(* IEC 61131-3 sources: AXOpen/src/components.rexroth.drives/ctrl/src (part 4) *)

(* ---- AxoIndraDriveAxisData.st ---- *)
NAMESPACE AXOpen.Components.Rexroth.Drives
    CLASS AxoIndraDriveAxisData
        VAR PUBLIC
            (* Commands *)
            CallAxis					:	BOOL;			//Call axis method for cyclic communication
            ReadOnlyData				:	BOOL;			//Read only data values from drive
            CallNumberCyclic			:	INT :=-1; 		//Number of method call's for cyclic communication
            WriteCommand				:	BOOL;			//Write command to drive
            PowerOnReq					:	BOOL;			//Request to power the drive on
            ResetReq					:	BOOL;			//Request to reset the drive
            HomingReq					:	BOOL;			//Request to start homing
            JogPositiveReq				:	BOOL;			//Request to jog the drive in positive direction
            JogNegativeReq				:	BOOL;			//Request to jog the drive in negative direction
            DriveStopReq				:	BOOL;			//Set Drive Stop with writing deceleration value to drive
            DriveHaltReq				:	BOOL;			//Set Drive Halt with writing deceleration value to drive
            MoveVelocityReq				:	BOOL;			//Command is velocity
            TorqueControlReq				:	BOOL;			//Command is torque
            Relative					:	BOOL; 			//Move relative to (last recommended) positioning command value
            Additive					:	BOOL; 			//Move additive to actual position; works only if relative possitioning active
            Position					:	LREAL;			//Target position for the motion  (negative or positive)
            Velocity					:	LREAL;			//Value of the maximum velocity (always positive) (not necessarily reached) [u/s].
            Acceleration				:	LREAL;			//Value of the acceleration (always positive) (increasing energy of the motor) [u/s2]
            Deceleration				:	LREAL;			//Value of the deceleration (always positive) (decreasing energy of the motor) [u/s2]
            Jerk						:	LREAL;			//Value of the jerk (always positive) [u/s3]
            Torque						:	LREAL;			//Value of the torque (always positive)
            S_0_0144_SignalStateWord	: 	WORD;			//S-0-0144 SignalStateWord*)
            CallAxisParameterMethod		:	BOOL;			//Call axis method for parameter read/write
            EnableAcyclicCommunication	:	BOOL;			//Enable acyclic communication (for parameter read/write)
            CallNumberAcyclic			:	INT;			//Number of method call's for acyclic communication
            WriteParameter				:	BOOL;			//FALSE = read, TRUE  = write Value of selected Parameter
            SelectDataType				:	UINT;			//0= Bool, 1 = Any, 2 = REAL
            ParameterNumber				:	DINT;			//Parameter number
            WriteValueDint				:	DINT;			//DINT value to be written
            WriteValueReal				:	REAL;			//REAL value to be written
            OverrideVelocityFactor		:	LREAL := 1.0;	//LREAL value to be written
            OverrideAccelerationFactor	:	LREAL := 1.0;	//LREAL value to be written
            OverrideJerkFactor			:	LREAL := 1.0;	//LREAL value to be written
        (* States *)
            CommandWriteActive			:	BOOL; 			//Command transfer to drive is active
            SetpointReached				: 	BOOL;			//Setpoint reached
            PowerOK						:	BOOL; 			//Power OK
            HomeOK						:	BOOL;			//Drive has reached the homeposition
            ResetOK						:	BOOL; 			//Reset done
            HomingRunning				:	BOOL;			//Homing is active
            Stopped						:	BOOL; 			//Drive in stopped regularly
            Standstill					:	BOOL; 			//Drive in standstill
            InPosition					:	BOOL; 			//Drive in position
            StoppedDueError				:	BOOL; 			//Drive in stop due to error
            MessageActive				:	BOOL;			//Class 3 diagnostics (message) present
            WarningActive				:	BOOL;			//Class 2 diagnostics (warning) present
            FailureActive				:	BOOL;			//Class 1 diagnostics (failure) present
            PowerError					:	BOOL; 			//Power-Failure
            StopError					:	BOOL;			//Stopping-Failure
            ContinuousMotion			:	BOOL; 			//Continius motion
            DiscreteMotion				:	BOOL; 			//Discrete motion
            SynchronizedMotion			:	BOOL;			//Synchronized motion
            Error						:	BOOL;			//Error
            ErrorID						:	AXOpen.Components.Rexroth.Drives.eAxoIndraDriveErrorCode;		//Error identification, ErrorCode
            ErrorIdent					:	AXOpen.Components.Rexroth.Drives.AxoIndraDriveErrorStruct;	//Error identification
            ActualPosition				:	LREAL; 			//Shows actual position
            ActualVelocity				:	LREAL; 			//Shows actual velocity
            ActualTorque				:	LREAL; 			//Shows actual torque
            CheckAccessOK				:	BOOL := TRUE;	//Flag for checking valid access at Axis_Data array
            S_0_0145_SignalControlWord	:	WORD;			//S-0-0145 wSignalControlWord, **** exept bit 0 *****)

            DoneAcyclicCommunication 	:	BOOL; 			//Reading/writing of the individual parameter completed, output variables valid
            ActiveAcyclicCommunication	: 	BOOL; 			//Reading/writing of the individual parameter active, output variables invalid
            DecimalPlaces 				:	UINT;			//Decimal places of the selected parameters
            DataTypeRead				:	UINT; 			//Read data type of the selected parameters
            DataLengthRead				:	UINT;			//Length of the read parameters
            ReadValueDint				:	DINT;			//DINT Operating value of the individual parameter without weighting
            ReadValueReal				:	REAL;			//REAL weighted operating value
            Error_AcyclicCommunication	:	BOOL := FALSE;  //Error
            ErrorID_AcyclicCommunication:   AXOpen.Components.Rexroth.Drives.eAxoIndraDriveErrorCode;		//Error identification, ErrorCode
            ErrorIdent_AcyclicCommunication:AXOpen.Components.Rexroth.Drives.AxoIndraDriveErrorStruct; 	//Error identification

        END_VAR

    END_CLASS

END_NAMESPACE

(* ---- AxoIndraDriveAxisReference.st ---- *)
// USING AXOpen.Components.Drives;

NAMESPACE AXOpen.Components.Rexroth.Drives
    CLASS AxoIndraDriveAxisReference IMPLEMENTS AXOpen.Components.Abstractions.Drives.IAxoAxisReference
        VAR PUBLIC
            FieldBus_In     :   AXOpen.Components.Rexroth.Drives.AxoIndraDriveFieldBusIn;
            FieldBus_Out    :   AXOpen.Components.Rexroth.Drives.AxoIndraDriveFieldBusOut;
            Parameter_In    :   AXOpen.Components.Rexroth.Drives.AxoIndraDriveParameterIn;
            Parameter_Out   :   AXOpen.Components.Rexroth.Drives.AxoIndraDriveParameterOut;
            Data            :   AXOpen.Components.Rexroth.Drives.AxoIndraDriveAxisData;
            Config          :   AXOpen.Components.Drives.AxoDrive_Config;
            Status          :   AXOpen.Components.Drives.AxoDrive_Status;
        END_VAR
    END_CLASS
END_NAMESPACE

(* ---- AxoIndraDriveFieldBusIn.st ---- *)
NAMESPACE AXOpen.Components.Rexroth.Drives
    CLASS AxoIndraDriveFieldBusIn
        (******************* Drive configuration  ***********************
        Master communication; Fieldbus settings:

                Profile type: * free configurable mode*
                    Configuration of realtime channel:
                        realtime input (configured feedback values):	    (9words)
                                P-0-4078 Fieldbus status WORD               (2bytes)
                                S-0-0051 Position feedback 1 value          (4bytes)
                                S-0-0040 Veloccity feedback value           (4bytes)
                                S-0-0390 Diagnostig message number          (4bytes)
                                S-0-0144 Signal status  word			    (2bytes)
                                S-0-0084 Actual torque/force value          (2bytes)
                        realtime output (configured command values):		(13words)
                                P-0-4077 Fieldbus control WORD              (2bytes)
                                S-0-0282 Positioning command value          (4bytes)
                                S-0-0259 Positioning velocity value         (4bytes)
                                S-0-0260 Positioning Accelelration          (4bytes)
                                S-0-0359 Positioning Deceleration           (4bytes)
                                S-0-0145 Signal control word                (2bytes)
                                S-0-0080 Torque/force command value		    (2bytes)
                                S-0-0193 Positioning jerk                   (4bytes)
                General settings:
                        S-0-0027, Configuration list signal control word -> Number 0; Content S-0-0393
                        S-0-0329, Assign list signal control word -> Number 0; Content 2
                        Primary operation mode: Drive controlled positioning, encoder 1 (without axis control word)
                        Secondary operation mode: Torque/force control
        *)
        VAR PUBLIC
            PhaseAcknowledgeBit0		:	BOOL;		//Operating mode acknowledge bit 0
            PhaseAcknowledgeBit1 		:	BOOL;		//Operating mode acknowledge bit 1
            InReference 				:	BOOL;		//In reference
            InStandstill 				:	BOOL;		//In standstill
            SetpointReached				:	BOOL;		//Setpoint reached
            CommandChangeBit 			:	BOOL;		//Command change bit
            OperatingModeError 			:	BOOL;		//Operating mode_error
            StatusSetpointProcess 		:	BOOL;		//Status setpoint processing
            ActualOperatingModeBit0 	:	BOOL;		//Actual_operating mode bit 0
            ActualOperatingModeBit1 	:	BOOL;		//Actual_operating mode bit 1
            SetpointAcknowledge 		:	BOOL;		//Setpoint acknowledge
            MessageZKL3 				:	BOOL;		//Message ZKL3
            WarningZKL2 				:	BOOL;		//Warning ZKL2
            DriveErrorZKL1 				:	BOOL;		//Drive Error ZKL1
            ReadyToOperateBit0 			:	BOOL;		//Ready to operate bit 0
            ReadyToOperateBit1 			:	BOOL;		//Ready to operate bit 1
            S_0_0051_ActualPosition		:	DWORD;		//Actual position
            S_0_0040_ActualVelocity		:	DWORD;		//Actual velocity
            S_0_0390_Diagnosis			:	DWORD;		//Diagnosis
            S_0_0144_SignalStatusWord	:	WORD;		//Signal status word
            S_0_0084_ActualTorque 		:	WORD;		//Actual torque
        END_VAR
    END_CLASS

END_NAMESPACE

(* ---- AxoIndraDriveFieldBusOut.st ---- *)
NAMESPACE AXOpen.Components.Rexroth.Drives
    CLASS AxoIndraDriveFieldBusOut
        (******************* Drive configuration  ***********************
        Master communication; Fieldbus settings:

                Profile type: * free configurable mode*
                    Configuration of realtime channel:
                        realtime input (configured feedback values):	    (9words)
                                P-0-4078 Fieldbus status WORD               (2bytes)
                                S-0-0051 Position feedback 1 value          (4bytes)
                                S-0-0040 Veloccity feedback value           (4bytes)
                                S-0-0390 Diagnostig message number          (4bytes)
                                S-0-0144 Signal status  word			    (2bytes)
                                S-0-0084 Actual torque/force value          (2bytes)
                        realtime output (configured command values):		(13words)
                                P-0-4077 Fieldbus control WORD              (2bytes)
                                S-0-0282 Positioning command value          (4bytes)
                                S-0-0259 Positioning velocity value         (4bytes)
                                S-0-0260 Positioning Accelelration          (4bytes)
                                S-0-0359 Positioning Deceleration           (4bytes)
                                S-0-0145 Signal control word                (2bytes)
                                S-0-0080 Torque/force command value		    (2bytes)
                                S-0-0193 Positioning jerk                   (4bytes)
                General settings:
                        S-0-0027, Configuration list signal control word -> Number 0; Content S-0-0393
                        S-0-0329, Assign list signal control word -> Number 0; Content 2
                        Primary operation mode: Drive controlled positioning, encoder 1 (without axis control word)
                        Secondary operation mode: Torque/force control
        *)
        VAR PUBLIC
            SetpointAcceptance 				:	BOOL;			//Setpoint acceptance
            OperatingModeSet 				:	BOOL;			//Operating mode set
            DriveToZeroPoint 				:	BOOL;			//Drive to zero point
            AbsoluteRelative 				:	BOOL;			//Position absolute = 0 or relative = 1
            ImmediateBlockChange 			:	BOOL;			//Immediate change
            ErrorDelete 					:	BOOL;			//Clear error
            JogForward 						:	BOOL;			//Jog forward
            JogBackward 					:	BOOL;			//Jog backward
            SetOperatingModeBit0 			:	BOOL;			//Setpoint operating mode_bit0
            SetOperatingModeBit1 			:	BOOL;			//Setpoint operating mode_bit1
            Iposync 						:	BOOL;			//Only in cycl. pos. control
            DriveHalt 						:	BOOL;			//Drive halt
            DriveEnable 					:	BOOL;			//Drive enable
            DriveOn 						:	BOOL;			//Drive on
            S_0_0282_CommandPosition		: 	DWORD;			//Command position
            S_0_0259_CommandVelocity		: 	DWORD;          //Command velocity
            S_0_0260_CommandAcceleration	: 	DWORD;          //Command acceleration
            S_0_0359_CommandDecceleration	: 	DWORD;          //Command decceleration
            S_0_0145_SignalControlWord		: 	WORD;           //Signal control word
            S_0_0080_TorqueForceCommand     :   WORD;           //Torque/force command value
            S_0_0193_CommandJerk            :   DWORD;          //Command jerk
        END_VAR
    END_CLASS
END_NAMESPACE

(* ---- AxoIndraDriveParameterIn.st ---- *)
NAMESPACE AXOpen.Components.Rexroth.Drives
    CLASS AxoIndraDriveParameterIn
        (******************* IndraDrive configuration  ***********************
        Master communication; Fieldbus settings:
        Parameter chanel 10Bytes / 5 Words I/O
        *)
        VAR PUBLIC
            Datalength	:	BYTE;	//Length of  transfer data*)
            FL_0		:	BOOL;	//Length userdata bit 0
            FL_1		:	BOOL;	//Length userdata bit 1
            FL_2		:	BOOL;	//Length userdata bit 2
            FL_3		:	BOOL;	//Length userdata bit 3
            ToggleBit	:	BOOL;	//Toggle bit
            LastBit		:	BOOL;	//Last bit
            Failure		:	BOOL;	//Failure while communication
            Reserve		:	BOOL;	//Reserve
            DataWord_0	:	WORD;	//Data WORD 0
            DataWord_1	:	WORD;	//Data word 1
            DataWord_2	:	WORD;	//Data word 2
            DataWord_3	:	WORD;	//Data word 3
        END_VAR
    END_CLASS
 END_NAMESPACE

(* ---- AxoIndraDriveParameterOut.st ---- *)
NAMESPACE AXOpen.Components.Rexroth.Drives
    CLASS AxoIndraDriveParameterOut
        (******************* IndraDrive configuration  ***********************
        Master communication; Fieldbus settings:
        Parameter chanel 10Bytes / 5 Words I/O
        *)
        VAR PUBLIC
            Datalength		:	BYTE := BYTE#04;//Length of transfer data
            FL_0			:	BOOL;			//Length userdata bit 0
            FL_1			:	BOOL;			//Length userdata bit 1
            FL_2			:	BOOL;			//Length userdata bit 2
            FL_3			:	BOOL;			//Length userdata bit 3
            ToggleBit		:	BOOL;			//Toggle bit
            LastBit			:	BOOL;			//Last bit
            Initalisation	:	BOOL := TRUE;	//Initialisation
            Reserve			:	BOOL;			//Reserve
            Index			:	WORD;			//Index number
            Subindex		:	BYTE;			//Subindex number
            Axis			:	BYTE;			//Axis number
            DataWord_0		:	WORD;			//Data word 0
            DataWord_1		:	WORD;			//Data word 1
        END_VAR
    END_CLASS
END_NAMESPACE

(* ---- AxoRexrothDrive.st ---- *)
USING AXOpen.Messaging.Static;
USING AXOpen.Messaging;
USING AXOpen.Core;
USING AXOpen.Components.Abstractions;
USING AXOpen.Components.Abstractions.AxoDrives;

NAMESPACE AXOpen.Components.Rexroth.Drives
    {#ix-attr:[Container(Layout.Wrap)]}
    CLASS PUBLIC AxoIndraDrive EXTENDS AXOpen.Components.Abstractions.AxoDrives.AxoDrive IMPLEMENTS AXOpen.Components.Abstractions.AxoDrives.IAxoDrive
        VAR PUBLIC
        END_VAR

        ///<summary>
		/// Restores this instance .
        ///</summary>
        METHOD PROTECTED OVERRIDE Restore: IAxoTask
            VAR
                _index : INT;
            END_VAR
            // Status.Action.Id := UINT#0;
            // Status.Error.Id  := UINT#0;
            // Status.CurrentJobName := '';
            // _Messenger.Restore();
            // _TaskMessenger.Restore();

            // ClearInspectionResultsTask.Restore();
            // TriggerTask.Restore();
            // ChangeJobByNameTask.Restore();
            // ChangeJobByNumberTask.Restore();

            // IF NOT AcquisitionStatus.ExposureComplete AND NOT InspectionStatus.Error THEN
            //     Status.Action.Id := UINT#300;
            //     RestoreTask.DoneWhen(TRUE);
            // END_IF;
            ;
        END_METHOD

        ///<summary>
		/// Custom logic for the manual control.
        ///</summary>
        METHOD PROTECTED OVERRIDE ManualControl
            // ChangeJobByNameTask.Manual(RequiredJobName);
            // ChangeJobByNumberTask.Manual(RequiredJobNumber);
            // SoftEventTask.Manual(RequiredSoftEventNumber);
            ;
        END_METHOD

        ///<summary>
        /// Ensures swapping the hardware input data structure into the AxisRef data structure
        ///</summary>
        METHOD PROTECTED OVERRIDE UpdateInputs : BOOL
            VAR_INPUT
                refAxisIn       :   REF_TO  ARRAY[*] OF BYTE;   //  Reference to the input data of the axis
            END_VAR
            VAR_IN_OUT
                AxisRef    :   AxoAxisRef;
            END_VAR
            ;
        END_METHOD

        ///<summary>
        /// Ensures swapping the AxisRef data structure into the hardware output data structure
        ///</summary>
        METHOD PROTECTED OVERRIDE UpdateOutputs : BOOL
            VAR_IN_OUT
                AxisRef    :   AxoAxisRef;
            END_VAR
            VAR_INPUT
                refAxisOut      :   REF_TO  ARRAY[*] OF BYTE;   //  Reference to the output data of the axis
            END_VAR
            ;
        END_METHOD

        ///<summary>
        /// This method controls the power stage (On or Off).
        ///</summary>
        METHOD PUBLIC OVERRIDE MC_Power
            VAR_IN_OUT
                AxisRef         :   AxoAxisRef;
            END_VAR
            VAR_INPUT
                Enable          :   BOOL;                       //  As long as ‘Enable’ is true, power is being enabled.
            END_VAR
            VAR_OUTPUT
                Status          :   BOOL;                       //  Effective state of the power stage
                Valid           :   BOOL;                       //  If true, a valid set of outputs is available at the method
                Error           :   BOOL;                       //  Signals that an error has occurred within the method
                ErrorID         :   WORD;                       //  Error identification
            END_VAR
            ;
        END_METHOD

        ///<summary>
        /// This method commands the axis to perform the «search home» sequence. The details of this sequence are
        /// manufacturer dependent and can be set by the axis’ parameters. The ‘Position’ input is used to set the absolute
        /// position when reference signal is detected. This method completes at ‘Standstill’ if it was started in ‘Standstill’.
        ///</summary>
        METHOD PUBLIC OVERRIDE MC_Home
            VAR_IN_OUT
                AxisRef         :   AxoAxisRef;                 //  Reference to the axis
            END_VAR
            VAR_INPUT
                Execute         :   BOOL;                       //  Start the motion at rising edge
                Position        :   LREAL;                      //  Absolute position when the reference signal is detected
                HommingMode     :   INT;                        //  Required homming mode
                Velocity        :   LREAL;                      //  Value of the maximum ‘Velocity’ (not necessarily reached) [u/s].
                Acceleration    :   LREAL;                      //  Value of the ‘Acceleration’ (always positive) (increasing energy of the motor) [u/s2]
                Deceleration    :   LREAL;                      //  Value of the ‘Deceleration’ (always positive) (decreasing energy of the motor) [u/s2]
            END_VAR
            VAR_OUTPUT
                Done            :   BOOL;                       // Reference known and set sucessfully
                Busy            :   BOOL;                       // The method is not finished and new output values are to be expected
                Active          :   BOOL;                       // Indicates that the method has control on the axis
                CommandAborted  :   BOOL;                       // ‘Command’ is aborted by another command
                Error           :   BOOL;                       // Signals that an error has occurred within the method
                ErrorID         :   WORD;                       // Error identification
             END_VAR
             ;
        END_METHOD

        ///<summary>
        /// This method commands a controlled motion stop and transfers the axis to the state ‘Stopping’. It aborts any
        /// ongoing method execution. While the axis is in state ‘Stopping’, no other method can perform any motion on the
        /// same axis.
        ///</summary>
        METHOD PUBLIC OVERRIDE MC_Stop
            VAR_IN_OUT
                AxisRef         :   AxoAxisRef;                 //  Reference to the axis
            END_VAR
            VAR_INPUT
                Execute         :   BOOL;                       //  Start the action at rising edge
                Deceleration    :   LREAL;                      //  Value of the ‘Deceleration’ [u/s2]
                Jerk            :   LREAL;                      //  Value of the ‘Jerk’ [u/s3]
            END_VAR
            VAR_OUTPUT
                Done            :   BOOL;                       // Zero velocity reached
                Busy            :   BOOL;                       // The method is not finished and new output values are to be expected
                Active          :   BOOL;                       // Indicates that the method has control on the axis
                CommandAborted  :   BOOL;                       // ‘Command’ is aborted by switching off power (only possibility to abort)
                Error           :   BOOL;                       // Signals that an error has occurred within the method
                ErrorID         :   WORD;                       // Error identification
             END_VAR
             ;
        END_METHOD

        ///<summary>
        /// This method commands a controlled motion stop. The axis is moved to the state ‘DiscreteMotion’, until the
        /// velocity is zero. With the ‘Done’ output set, the state is transferred to ‘Standstill’.
        ///</summary>
        METHOD PUBLIC OVERRIDE MC_Halt
            VAR_IN_OUT
                AxisRef         :   AxoAxisRef;                 //  Reference to the axis
            END_VAR
            VAR_INPUT
                Execute         :   BOOL;                       //  Start the action at rising edge
                Deceleration    :   LREAL;                      //  Value of the ‘Deceleration’ [u/s2]
                Jerk            :   LREAL;                      //  Value of the ‘Jerk’ [u/s3]
            END_VAR
            VAR_OUTPUT
                Done            :   BOOL;                       // Zero velocity reached
                Busy            :   BOOL;                       // The method is not finished and new output values are to be expected
                Active          :   BOOL;                       // Indicates that the method has control on the axis
                CommandAborted  :   BOOL;                       // ‘Command’ is aborted by switching off power (only possibility to abort)
                Error           :   BOOL;                       // Signals that an error has occurred within the method
                ErrorID         :   WORD;                       // Error identification
             END_VAR
             ;
        END_METHOD

        ///<summary>
        /// This method commands a controlled motion to a specified absolute position.
        ///<summary>
        METHOD PUBLIC OVERRIDE MC_MoveAbsolute
            VAR_IN_OUT
                AxisRef         :   AxoAxisRef;                 //  Reference to the axis
            END_VAR
            VAR_INPUT
                Execute         :   BOOL;                       //  Start the motion at rising edge
                ContinuousUpdate:   BOOL;                       //  Activate ‘ContinuousUpdate’ - target parameters should be changed during movement
                Position        :   LREAL;                      //  Commanded ‘Position’ for the motion (in technical unit [u]) (negative or positive)
                Velocity        :   LREAL;                      //  Value of the maximum ‘Velocity’ (not necessarily reached) [u/s].
                Acceleration    :   LREAL;                      //  Value of the ‘Acceleration’ (always positive) (increasing energy of the motor) [u/s2]
                Deceleration    :   LREAL;                      //  Value of the ‘Deceleration’ (always positive) (decreasing energy of the motor) [u/s2]
                Jerk            :   LREAL;                      //  Value of the ‘Jerk’ [u/s3]
                Direction       :   eAxoDriveDirection;         //  Enum type (1-of-4 values: PositiveDirection, ShortestWay, NegativeDirection, CurrentDirection)
            END_VAR
            VAR_OUTPUT
                Done            :   BOOL;                       // Commanded position finally reached
                Busy            :   BOOL;                       // The method is not finished and new output values are to be expected
                Active          :   BOOL;                       // Indicates that the method has control on the axis
                CommandAborted  :   BOOL;                       // ‘Command’ is aborted by another command
                Error           :   BOOL;                       // Signals that an error has occurred within the method
                ErrorID         :   WORD;                       // Error identification
             END_VAR
             ;
        END_METHOD

        ///<summary>
        /// This method  commands a controlled motion of a specified distance relative to the set position at the time of the execution.
        ///<summary>
        METHOD PUBLIC OVERRIDE MC_MoveRelative
            VAR_IN_OUT
                AxisRef         :   AxoAxisRef;                 //  Reference to the axis
            END_VAR
            VAR_INPUT
                Execute         :   BOOL;                       //  Start the motion at rising edge
                ContinuousUpdate:   BOOL;                       //  Activate ‘ContinuousUpdate’ - target parameters should be changed during movement
                Distance        :   LREAL;                      //  Relative distance for the motion (in technical unit [u]
                Velocity        :   LREAL;                      //  Value of the maximum ‘Velocity’ (not necessarily reached) [u/s].
                Acceleration    :   LREAL;                      //  Value of the ‘Acceleration’ (always positive) (increasing energy of the motor) [u/s2]
                Deceleration    :   LREAL;                      //  Value of the ‘Deceleration’ (always positive) (decreasing energy of the motor) [u/s2]
                Jerk            :   LREAL;                      //  Value of the ‘Jerk’ [u/s3]
                Direction       :   eAxoDriveDirection;         //  Enum type (1-of-4 values: PositiveDirection, ShortestWay, NegativeDirection, CurrentDirection)
            END_VAR
            VAR_OUTPUT
                Done            :   BOOL;                       // Commanded distance reached
                Busy            :   BOOL;                       // The method is not finished and new output values are to be expected
                Active          :   BOOL;                       // Indicates that the method has control on the axis
                CommandAborted  :   BOOL;                       // ‘Command’ is aborted by another command
                Error           :   BOOL;                       // Signals that an error has occurred within the method
                ErrorID         :   WORD;                       // Error identification
             END_VAR
             ;
        END_METHOD

        ///<summary>
        /// This method commands a controlled motion of a specified relative distance additional to the most recent
        /// commanded position in the axis state ‘DiscreteMotion’. The most recent commanded position may be the result of a
        /// previous MC_MoveAdditive motion which was aborted. If the method is activated in the axis state ‘ContinuousMotion’, the
        /// specified relative distance is added to the set position at the time of the execution.
        ///<summary>
        METHOD PUBLIC OVERRIDE MC_MoveAdditive
            VAR_IN_OUT
                AxisRef         :   AxoAxisRef;                 //  Reference to the axis
            END_VAR
            VAR_INPUT
                Execute         :   BOOL;                       //  Start the motion at rising edge
                ContinuousUpdate:   BOOL;                       //  Activate ‘ContinuousUpdate’ - target parameters should be changed during movement
                Distance        :   LREAL;                      //  Relative distance for the motion (in technical unit [u]
                Velocity        :   LREAL;                      //  Value of the maximum ‘Velocity’ (not necessarily reached) [u/s].
                Acceleration    :   LREAL;                      //  Value of the ‘Acceleration’ (always positive) (increasing energy of the motor) [u/s2]
                Deceleration    :   LREAL;                      //  Value of the ‘Deceleration’ (always positive) (decreasing energy of the motor) [u/s2]
                Jerk            :   LREAL;                      //  Value of the ‘Jerk’ [u/s3]
                Direction       :   eAxoDriveDirection;         //  Enum type (1-of-4 values: PositiveDirection, ShortestWay, NegativeDirection, CurrentDirection)
            END_VAR
            VAR_OUTPUT
                Done            :   BOOL;                       // Commanded distance reached
                Busy            :   BOOL;                       // The method is not finished and new output values are to be expected
                Active          :   BOOL;                       // Indicates that the method has control on the axis
                CommandAborted  :   BOOL;                       // ‘Command’ is aborted by another command
                Error           :   BOOL;                       // Signals that an error has occurred within the method
                ErrorID         :   WORD;                       // Error identification
             END_VAR
             ;
        END_METHOD

        ///<summary>
        /// This method commands a never ending controlled motion at a specified velocity.
        ///<summary>
        METHOD PUBLIC OVERRIDE MC_MoveVelocity
            VAR_IN_OUT
                AxisRef         :   AxoAxisRef;                 //  Reference to the axis
            END_VAR
            VAR_INPUT
                Execute         :   BOOL;                       //  Start the motion at rising edge
                ContinuousUpdate:   BOOL;                       //  Activate ‘ContinuousUpdate’ - target parameters should be changed during movement
                Velocity        :   LREAL;                      //  Value of the maximum velocity [u/s]. Can be a signed value.
                Acceleration    :   LREAL;                      //  Value of the ‘Acceleration’ (always positive) (increasing energy of the motor) [u/s2]
                Deceleration    :   LREAL;                      //  Value of the ‘Deceleration’ (always positive) (decreasing energy of the motor) [u/s2]
                Jerk            :   LREAL;                      //  Value of the ‘Jerk’ [u/s3]
                Direction       :   eAxoDriveDirection;         //  Enum type (1-of-3 values: PositiveDirection, NegativeDirection, and CurrentDirection. Note: shortest way not applicable)
            END_VAR
            VAR_OUTPUT
                InVelocity      :   BOOL;                       // Commanded velocity reached
                Busy            :   BOOL;                       // The method is not finished and new output values are to be expected
                Active          :   BOOL;                       // Indicates that the method has control on the axis
                CommandAborted  :   BOOL;                       // ‘Command’ is aborted by another command
                Error           :   BOOL;                       // Signals that an error has occurred within the method
                ErrorID         :   WORD;                       // Error identification
             END_VAR
             ;
        END_METHOD

        ///<summary>
        /// This method continuously exerts a torque or force of the specified magnitude. This magnitude is
        /// approached using a defined ramp (‘TorqueRamp’), and the method sets the ‘InTorque’ output if the
        /// commanded torque level is reached. This method is applicable for force and torque. When there is no external
        /// load, force is applicable. Positive torque is in the positive direction of velocity.
        ///<summary>
        METHOD PUBLIC OVERRIDE MC_TorqueControl
            VAR_IN_OUT
                AxisRef         :   AxoAxisRef;                 //  Reference to the axis
            END_VAR
            VAR_INPUT
                Execute         :   BOOL;                       //  Start the motion at rising edge
                ContinuousUpdate:   BOOL;                       //  Activate ‘ContinuousUpdate’ - target parameters should be changed during movement
                Torque          :   LREAL;                      //  Value of the torque (Torque or force in technical unit [u])
                TorqueRamp      :   LREAL;                      //  The maximum time derivative of the set value of the torque or force (in technical unit per sec. [u/s])
                Velocity        :   LREAL;                      //  Absolute value of the maximum velocity.
                Acceleration    :   LREAL;                      //  Value of the maximum acceleration (acceleration is applicable with same sign of torque and velocity)
                Deceleration    :   LREAL;                      //  Value of the maximum deceleration (deceleration is applicable with opposite signs of torque and velocity)
                Jerk            :   LREAL;                      //  Value of the maximum jerk
                Direction       :   eAxoDriveDirection;         //  Enum type (1 of 2 values: PositiveDirection, NegativeDirection or CurrentDirection). Specifies the direction of the torque. (Note: Torque input can be signed value).
            END_VAR
            VAR_OUTPUT
                InTorque        :   BOOL;                       //  Setpoint value of torque or force equals the commandedvalue
                Busy            :   BOOL;                       //  The method is not finished and new output values are to be expected
                Active          :   BOOL;                       //  Indicates that the method has control on the axis
                CommandAborted  :   BOOL;                       //  ‘Command’ is aborted by another command
                Error           :   BOOL;                       //  Signals that an error has occurred within the method
                ErrorID         :   WORD;                       //  Error identification
            END_VAR
            ;
        END_METHOD

        ///<summary>
        /// This method shifts the coordinate system of an axis by manipulating both the set-point position as well as the
        /// actual position of an axis with the same value without any movement caused. (Re-calibration with same following error).
        /// This can be used for instance for a reference situation. This method can also be used during motion without changing
        /// the commanded position, which is now positioned in the shifted coordinate system.
        ///<summary>
        METHOD PUBLIC OVERRIDE MC_SetPosition
            VAR_IN_OUT
                AxisRef         :   AxoAxisRef;                 //  Reference to the axis
            END_VAR
            VAR_INPUT
                Execute         :   BOOL;                       //  Start setting position in axis
                Position        :   REAL;                       //  Position unit [u] (Means ‘Distance’ if ‘Relative’= TRUE)
                Relative        :   BOOL;                       //  ‘Relative’ distance if True, ‘Absolute’ position if False (= Default)
                ExecutionMode   :   eAxoExecutionMode;          //  Defines the chronological sequence of the method.
            END_VAR
            VAR_OUTPUT
                Done            :   BOOL;                       //  ‘Position’ has new value
                Error           :   BOOL;                       //  Signals that an error has occurred within the method
                ErrorID         :   WORD;                       //  Error identification
            END_VAR
            ;
        END_METHOD

        ///<summary>
        /// This method sets the values of override for the whole axis, and all functions that are working on that axis. The override
        /// parameters contribute as a factor to the calculation of the commanded velocity, acceleration and jerk of the motion.
        ///<summary>
        METHOD PUBLIC OVERRIDE MC_SetOverride
            VAR_IN_OUT
                AxisRef         :   AxoAxisRef;                 //  Reference to the axis
            END_VAR
            VAR_INPUT
                Enable          :   BOOL;                       //  If SET, it writes the value of the override factor continuously. If RESET it should keep the last value.
                VelFactor       :   LREAL;                      //  New override factor for the velocity
                AccFactor       :   LREAL;                      //  New override factor for the acceleration/deceleration
                JerkFactor      :   LREAL;                      //  New override factor for the jer
            END_VAR
            VAR_OUTPUT
                Enabled         :   BOOL;                       //  Signals that the override factor(s) is (are) set successfully
                Busy            :   BOOL;                       //  The method is not finished and new output values are to be expected
                Error           :   BOOL;                       //  Signals that an error has occurred within the method
                ErrorID         :   WORD;                       //  Error identification
            END_VAR
            ;
        END_METHOD

        ///<summary>
        /// This method returns the value of a vendor specific parameter. The returned Value has to be converted to Real
        /// if necessary. If not possible, the vendor has to supply a vendor specific method to read the parameter.
        ///<summary>
        METHOD PUBLIC OVERRIDE MC_ReadParameter
            VAR_IN_OUT
                AxisRef         :   AxoAxisRef;                 //  Reference to the axis
            END_VAR
            VAR_INPUT
                Enable          :   BOOL;                       //  Get the value of the parameter continuously while enabled
                ParameterNumber :   INT;                        //  Number of the parameter. One can also use symbolic parameter names which are declared as VAR CONST.
            END_VAR
            VAR_OUTPUT
                Valid           :   BOOL;                       //  A valid output is available at the method
                Busy            :   BOOL;                       //  The method is not finished and new output values are to be expected
                Error           :   BOOL;                       //  Signals that an error has occurred within the method
                ErrorID         :   WORD;                       //  Error identification
                Value           :   REAL;                       //  Value of the specified parameter in the datatype, as specified by the vendor
            END_VAR
            ;
        END_METHOD

        ///<summary>
        /// This method returns the value of a vendor specific parameter with datatype BOOL.
        ///<summary>
        METHOD PUBLIC OVERRIDE MC_ReadBoolParameter
            VAR_IN_OUT
                AxisRef         :   AxoAxisRef;                 //  Reference to the axis
            END_VAR
            VAR_INPUT
                Enable          :   BOOL;                       //  Get the value of the parameter continuously while enabled
                ParameterNumber :   INT;                        //  Number of the parameter. One can also use symbolic parameter names which are declared as VAR CONST.
            END_VAR
            VAR_OUTPUT
                Valid           :   BOOL;                       //  A valid output is available at the method
                Busy            :   BOOL;                       //  The method is not finished and new output values are to be expected
                Error           :   BOOL;                       //  Signals that an error has occurred within the method
                ErrorID         :   WORD;                       //  Error identification
                Value           :   BOOL;                       //  Value of the specified parameter in the datatype, as specified by the vendor
            END_VAR
            ;
        END_METHOD

        ///<summary>
        /// This method modifies the value of a vendor specific parameter.
        ///<summary>
        METHOD PUBLIC OVERRIDE MC_WriteParameter
            VAR_IN_OUT
                AxisRef         :   AxoAxisRef;                 //  Reference to the axis
            END_VAR
            VAR_INPUT
                Execute         :   BOOL;                       //  Write the value of the parameter at rising edge
                ParameterNumber :   INT;                        //  Number of the parameter (correspondence between number andparameter is specified in the table above)
                Value           :   REAL;                       //  New value of the specified parameter
                ExecutionMode   :   eAxoExecutionMode;          //  Defines the chronological sequence of the method.
            END_VAR
            VAR_OUTPUT
                Done            :   BOOL;                       //  Parameter successfully written
                Busy            :   BOOL;                       //  The method is not finished and new output values are to be expected.
                Error           :   BOOL;                       //  Signals that an error has occurred within the method
                ErrorID         :   WORD;                       //  Error identification
            END_VAR
            ;
        END_METHOD

        ///<summary>
        /// This method modifies the value of a vendor specific parameter of type BOOL.
        ///<summary>
        METHOD PUBLIC OVERRIDE MC_WriteBoolParameter
            VAR_IN_OUT
                AxisRef         :   AxoAxisRef;                 //  Reference to the axis
            END_VAR
            VAR_INPUT
                Execute         :   BOOL;                       //  Write the value of the parameter at rising edge
                ParameterNumber :   INT;                        //  Number of the parameter (correspondence between number andparameter is specified in the table above)
                Value           :   BOOL;                       //  New value of the specified parameter
                ExecutionMode   :   eAxoExecutionMode;          //  Defines the chronological sequence of the method.
            END_VAR
            VAR_OUTPUT
                Done            :   BOOL;                       //  Parameter successfully written
                Busy            :   BOOL;                       //  The method is not finished and new output values are to be expected.
                Error           :   BOOL;                       //  Signals that an error has occurred within the method
                ErrorID         :   WORD;                       //  Error identification
            END_VAR
            ;
        END_METHOD

        ///<summary>
        /// This method gives access to the value of the input, referenced by the datatype MC_INPUT_REF.
        /// It provides the value of the referenced input (BOOL).
        ///<summary>
        METHOD PUBLIC OVERRIDE MC_ReadDigitalInput
            VAR_IN_OUT
                AxisRef         :   AxoAxisRef;                 //  Reference to the axis
            END_VAR
            VAR_INPUT
                Enable          :   BOOL;                       //  Get the value of the selected input signal continuously while enabled
                InputNumber     :   INT;                        //  Selects the input. Can be part of MC_INPUT_REF, if only one single input is referenced.
            END_VAR
            VAR_OUTPUT
                Valid           :   BOOL;                       //  A valid output is available at the method
                Busy            :   BOOL;                       //  The method is not finished and new output values are to be expected
                Error           :   BOOL;                       //  Signals that an error has occurred within the method
                ErrorID         :   WORD;                       //  Error identification
                Value           :   BOOL;                       //  The value of the selected input signal
            END_VAR
            ;
        END_METHOD

        ///<summary>
        /// This method provides access to the value of a digital output, referenced by the datatype MC_OUTPUT_REF.
        /// It provides the value of the referenced output (BOOL).
        ///<summary>
        METHOD PUBLIC OVERRIDE MC_ReadDigitalOutput
            VAR_IN_OUT
                AxisRef         :   AxoAxisRef;                 //  Reference to the axis
            END_VAR
            VAR_INPUT
                Enable          :   BOOL;                       //  Get the value of the selected output signal continuously while enabled
                OutputNumber    :   INT;                        //  Selects the output. Can be part of MC_OUTPUT_REF, if only one single output is referenced.
            END_VAR
            VAR_OUTPUT
                Valid           :   BOOL;                       //  A valid output is available at the method
                Busy            :   BOOL;                       //  The method is not finished and new output values are to be expected
                Error           :   BOOL;                       //  Signals that an error has occurred within the method
                ErrorID         :   WORD;                       //  Error identification
                Value           :   BOOL;                       //  The value of the selected output signal
            END_VAR
            ;
        END_METHOD

        ///<summary>
        /// This method writes a value to the output referenced by the argument ‘Output’ once (with rising edge of Execute)
        ///<summary>
        METHOD PUBLIC OVERRIDE MC_WriteDigitalOutput
            VAR_IN_OUT
                AxisRef         :   AxoAxisRef;                 //  Reference to the axis
            END_VAR
            VAR_INPUT
                Enable          :   BOOL;                       //  Get the value of the selected output signal continuously while enabled
                OutputNumber    :   INT;                        //  Selects the output. Can be part of MC_OUTPUT_REF, if only one single output is referenced.
                Value           :   BOOL;                       //  The value of the selected output signal
                ExecutionMode   :   eAxoExecutionMode;          //  Defines the chronological sequence of the method.
            END_VAR
            VAR_OUTPUT
                Done            :   BOOL;                       //  Writing of the output signal value is done
                Busy            :   BOOL;                       //  The method is not finished and new output values are to be expected.
                Error           :   BOOL;                       //  Signals that an error has occurred within the method
                ErrorID         :   WORD;                       //  Error identification
            END_VAR
            ;
        END_METHOD

        ///<summary>
        /// This method returns the actual position.
        ///<summary>
        METHOD PUBLIC OVERRIDE MC_ReadActualPosition
            VAR_IN_OUT
                AxisRef         :   AxoAxisRef;                 //  Reference to the axis
            END_VAR
            VAR_INPUT
                Enable          :   BOOL;                       //  Get the value of the parameter continuously while enabled
            END_VAR
            VAR_OUTPUT
                Valid           :   BOOL;                       //  A valid output is available at the method
                Busy            :   BOOL;                       //  The method is not finished and new output values are to be expected
                Error           :   BOOL;                       //  Signals that an error has occurred within the method
                ErrorID         :   WORD;                       //  Error identification
                Position        :   REAL;                       //  New absolute position (in axis’ unit [u])
            END_VAR
            ;
        END_METHOD

        ///<summary>
        /// This method returns the value of the actual velocity as long as ‘Enable’ is set. ‘Valid’ is true when the
        /// dataoutput ‘Velocity’ is valid. If ‘Enable’ is Reset, the data loses its validity, and all outputs are reset,
        /// no matter if new data is available.
        ///<summary>
        METHOD PUBLIC OVERRIDE MC_ReadActualVelocity
            VAR_IN_OUT
                AxisRef         :   AxoAxisRef;                 //  Reference to the axis
            END_VAR
            VAR_INPUT
                Enable          :   BOOL;                       //  Get the value of the parameter continuously while enabled
            END_VAR
            VAR_OUTPUT
                Valid           :   BOOL;                       //  A valid output is available at the method
                Busy            :   BOOL;                       //  The method is not finished and new output values are to be expected
                Error           :   BOOL;                       //  Signals that an error has occurred within the method
                ErrorID         :   WORD;                       //  Error identification
                Velocity        :   REAL;                       //  The value of the actual velocity (in axis’ unit [u/s])
            END_VAR
            ;
        END_METHOD

        ///<summary>
        /// This method returns the value of the actual torque or force as long as ‘Enable’ is set. ‘Valid’ is true when the
        /// data-output ‘Torque’ is valid. If ‘Enable’ is Reset, the data loses its validity, and ‘Valid’ is also reset,
        /// no matter if new data is available.
        ///<summary>
        METHOD PUBLIC OVERRIDE MC_ReadActualTorque
            VAR_IN_OUT
                AxisRef         :   AxoAxisRef;                 //  Reference to the axis
            END_VAR
            VAR_INPUT
                Enable          :   BOOL;                       //  Get the value of the parameter continuously while enabled
            END_VAR
            VAR_OUTPUT
                Valid           :   BOOL;                       //  A valid output is available at the method
                Busy            :   BOOL;                       //  The method is not finished and new output values are to be expected
                Error           :   BOOL;                       //  Signals that an error has occurred within the method
                ErrorID         :   WORD;                       //  Error identification
                Torque          :   REAL;                       //  The value of the actual torque or force (in technical units)
            END_VAR
            ;
        END_METHOD

        ///<summary>
        /// This method returns in detail the status of the state diagram of the axis
        ///<summary>
        METHOD PUBLIC OVERRIDE MC_ReadStatus
            VAR_IN_OUT
                AxisRef         :   AxoAxisRef;                 //  Reference to the axis
            END_VAR
            VAR_INPUT
                Enable          :   BOOL;                       //  Get the value of the parameter continuously while enabled
            END_VAR
            VAR_OUTPUT
                Valid           :   BOOL;                       //  A valid output is available at the method
                Busy            :   BOOL;                       //  The method is not finished and new output values are to be expected
                Error           :   BOOL;                       //  Signals that an error has occurred within the method
                ErrorID         :   WORD;                       //  Error identification
                ErrorStop       :   BOOL;                       //  See state diagram
                Disabled        :   BOOL;                       //  See state diagram
                Stopping        :   BOOL;                       //  See state diagram
                Homing          :   BOOL;                       //  See state diagram
                Standstill      :   BOOL;                       //  See state diagram
                DiscreteMotion  :   BOOL;                       //  See state diagram
                ContinuousMotion:   BOOL;                       //  See state diagram
                SynchronizedMotion: BOOL;                       //  See state diagram
            END_VAR
            ;
        END_METHOD

        ///<summary>
        /// This method returns in detail the status of the axis with respect to the motion currently in progress.
        ///<summary>
        METHOD PUBLIC OVERRIDE MC_ReadMotionState
            VAR_IN_OUT
                AxisRef         :   AxoAxisRef;                 //  Reference to the axis
            END_VAR
            VAR_INPUT
                Enable          :   BOOL;                       //  Get the value of the parameter continuously while enabled
                Source          :   eAxoSource;                 //  Defines the source of the relevant data: CommandedValue;SetValue, ActualValue.
            END_VAR
            VAR_OUTPUT
                Valid           :   BOOL;                       //  A valid output is available at the method
                Busy            :   BOOL;                       //  The method is not finished and new output values are to be expected
                Error           :   BOOL;                       //  Signals that an error has occurred within the method
                ErrorID         :   WORD;                       //  Error identification
                ConstantVelocity:   BOOL;                       //  Velocity is constant. Velocity may be 0. For the actual value a window is applicable (window is vendor specific)
                Accelerating    :   BOOL;                       //  Increasing the absolute value of the velocity
                Decelerating    :   BOOL;                       //  Decreasing the absolute value of the velocity
                DirectionPositive:  BOOL;                       //  Signals that the position is increasing
                DirectionNegative:  BOOL;                       //  Signals that the position is decreasing
            END_VAR
            ;
        END_METHOD

        ///<summary>
        /// This method reads information concerning an axis, like modes, inputs directly related to the axis,
        /// and certain status information.
        ///<summary>
        METHOD PUBLIC OVERRIDE MC_ReadAxisInfo
            VAR_IN_OUT
                AxisRef         :   AxoAxisRef;                 //  Reference to the axis
            END_VAR
            VAR_INPUT
                Enable          :   BOOL;                       //  Get the value of the parameter continuously while enabled
            END_VAR
            VAR_OUTPUT
                Valid           :   BOOL;                       //  A valid output is available at the method
                Busy            :   BOOL;                       //  The method is not finished and new output values are to be expected
                Error           :   BOOL;                       //  Signals that an error has occurred within the method
                ErrorID         :   WORD;                       //  Error identification
                HomeAbsSwitch   :   BOOL;                       //  Digital home switch input is active
                LimitSwitchPos  :   BOOL;                       //  Positive hardware end switch is active
                LimitSwitchNeg  :   BOOL;                       //  Negative hardware end switch is active
                Simulation      :   BOOL;                       //  Axis is in simulation mode (e.g. motor is simulated)
                CommunicationReady: BOOL;                       //  “Network” is initialized and ready for communication
                ReadyForPowerOn :   BOOL;                       //  Drive is ready to be enabled (power on)
                PowerOn         :   BOOL;                       //  If TRUE shows that the power stage is switched ON
                IsHomed         :   BOOL;                       //  The absolute reference position is known for the axis (axis is homed)
                AxisWarning     :   BOOL;                       //  Warning(s) on the axis is present
            END_VAR
            ;
        END_METHOD

        ///<summary>
        /// This method presents general axis errors not relating to the methods.
        /// (for instance axis errors, drive errors, communication errors)
        ///<summary>
        METHOD PUBLIC OVERRIDE MC_ReadAxisError
            VAR_IN_OUT
                AxisRef         :   AxoAxisRef;                 //  Reference to the axis
            END_VAR
            VAR_INPUT
                Enable          :   BOOL;                       //  Get the value of the parameter continuously while enabled
            END_VAR
            VAR_OUTPUT
                Valid           :   BOOL;                       //  A valid output is available at the method
                Busy            :   BOOL;                       //  The method is not finished and new output values are to be expected
                Error           :   BOOL;                       //  Signals that an error has occurred within the method
                ErrorID         :   WORD;                       //  Error identification
                AxisErrorID     :   WORD;                       //  The value of the axis error. These values are vendor specific
            END_VAR
            ;
        END_METHOD

        ///<summary>
        /// This method makes the transition from the state ‘ErrorStop’ to ‘Standstill’ or ‘Disabled’ by resetting all
        /// internal axis-related errors – it does not affect the output of the other methods.
        ///<summary>
        METHOD PUBLIC OVERRIDE MC_Reset
            VAR_IN_OUT
                AxisRef         :   AxoAxisRef;                 //  Reference to the axis
            END_VAR
            VAR_INPUT
                Execute         :   BOOL;                       //  Resets all internal axis-related error
            END_VAR
            VAR_OUTPUT
                Done            :   BOOL;                       //  ‘Standstill’ or ‘Disabled’ state is reached
                Busy            :   BOOL;                       //  The method is not finished and new output values are to be expected
                Error           :   BOOL;                       //  Signals that an error has occurred within the method
                ErrorID         :   WORD;                       //  Error identification
            END_VAR
            ;
        END_METHOD
    END_CLASS

END_NAMESPACE

(* ---- Cylinder.st ---- *)
USING AXOpen.Core;
USING AXOpen.Messaging;
USING AXOpen.Messaging.Static;

NAMESPACE AXOpen.Pneumatics
    CLASS Cylinder EXTENDS AXOpen.Core.AxoComponent
        VAR PUBLIC
            {#ix-attr:[Container(Layout.Wrap)]}
            {#ix-attr:[ComponentHeader()]}
            MoveToWork : AxoTask;
            {#ix-attr:[ComponentHeader()]}
            MoveToHome : AxoTask;

            {#ix-attr:[ComponentDetails("Tasks")]}
            Stop : AxoTask;

            {#ix-attr:[Container(Layout.Stack)]}
            {#ix-attr:[ComponentDetails("Signals")]}
            {#ix-attr:[ReadOnly()]}
            {#ix-set:AttributeName = "<#Home sensor#>"}
            _HomeSensor : BOOL;
            {#ix-attr:[ComponentDetails("Signals")]}
            {#ix-attr:[ReadOnly()]}
            {#ix-set:AttributeName = "<#Work sensor#>"}
            _WorkSensor : BOOL;
            {#ix-attr:[Container(Layout.Stack)]}
            {#ix-attr:[ComponentDetails("Signals")]}
            {#ix-attr:[ReadOnly()]}
            {#ix-set:AttributeName = "<#Move home signal#>"}
            _MoveHomeSignal : BOOL;
            {#ix-attr:[ComponentDetails("Signals")]}
            {#ix-attr:[ReadOnly()]}
            {#ix-set:AttributeName = "<#Move work signal#>"}
            _MoveWorkSignal : BOOL;

            {#ix-set:MessageText = "<#Movement to work position did not succeed.#>"}
            {#ix-set:Help = "<#Check the cyclinder that it is free to move, air pressure input and extremity sensor.#>"}
            _MoveToWorkNotReached : AXOpen.Messaging.Static.AxoMessenger;

            {#ix-set:MessageText = "<#Movement to home position did not succeed.#>"}
            {#ix-set:Help = "<#Check the cyclinder that it is free to move, air pressure input and extremity sensor.#>"}
            _MoveToHomeNotReached : AXOpen.Messaging.Static.AxoMessenger;
        END_VAR

        ///<summary>
        /// Runs tasks and logic of this component.
        /// >[!IMPORTANT] This method must or one of its overloads be called cyclically.
        ///</summary>
        METHOD PUBLIC Run
            VAR_INPUT
                parent : IAxoObject;
                homeSensor : BOOL;
                workSensor : BOOL;
            END_VAR
            VAR_OUTPUT
                moveHomeSignal : BOOL;
                moveWorkSignal : BOOL;
            END_VAR
            IF (parent = NULL) THEN RETURN; END_IF;
            THIS.Initialize(parent);
            THIS.Run(parent.GetContext(), homeSensor, workSensor, moveHomeSignal, moveWorkSignal);
        END_METHOD

        ///<summary>
        /// Runs tasks and logic of this component.
        /// >[!IMPORTANT] This method must or one of its overloads be called cyclically.
        ///</summary>
        METHOD PUBLIC Run
            VAR_INPUT
                context : IAxoContext;
                homeSensor : BOOL;
                workSensor : BOOL;
            END_VAR
            VAR_OUTPUT
                moveHomeSignal : BOOL;
                moveWorkSignal : BOOL;
            END_VAR

            THIS.Open();

            THIS.Initialize(context);
            MoveToWork.Initialize(THIS);
            MoveToHome.Initialize(THIS);
            Stop.Initialize(THIS);

            _MoveToWorkNotReached.Serve(THIS);
            _MoveToHomeNotReached.Serve(THIS);

            IF(Stop.Execute()) THEN
                moveHomeSignal := FALSE;
                moveWorkSignal := FALSE;
                MoveToHome.Restore();
                MoveToWork.Restore();
                Stop.DoneWhen(TRUE);
                Stop.Restore();
            END_IF;

            IF(MoveToWork.Execute()) THEN
                moveHomeSignal := FALSE;
                moveWorkSignal := TRUE;
                MoveToWork.DoneWhen(workSensor);
                MoveToHome.Restore();

                _MoveToWorkNotReached.ActivateOnCondition(MoveToWork.Duration >= T#10S, eAxoMessageCategory#Error);
            END_IF;

            IF(MoveToHome.Execute()) THEN
                moveHomeSignal := TRUE;
                moveWorkSignal := FALSE;
                MoveToHome.DoneWhen(homeSensor);
                MoveToWork.Restore();
                _MoveToHomeNotReached.ActivateOnCondition(MoveToHome.Duration >= T#10S, eAxoMessageCategory#Error);
            END_IF;

            _HomeSensor := homeSensor;
            _WorkSensor := workSensor;

            _MoveHomeSignal := moveHomeSignal;
            _MoveWorkSignal := moveWorkSignal;

            THIS.Close();
        END_METHOD

        METHOD PROTECTED OVERRIDE ManualControl
            THIS._isManuallyControllable := true;
        END_METHOD

        ///<summary>
        /// Restores this component into intial state.
        ///</summary>
        METHOD PROTECTED OVERRIDE Restore : IAxoTask
            MoveToWork.Restore();
            MoveToWork.Restore();
            Stop.Restore();
        END_METHOD
    END_CLASS
END_NAMESPACE
